// TIA Portal V20 export
FUNCTION_BLOCK "ErrComTextList"   // FB305, FBD
{ S7_Optimized_Access := 'TRUE' }
// stored: AutoNumber false, MemoryReserve 100, SetENOAutomatically false
   VAR
      Var { ExternalAccessible := 'False'; ExternalVisible := 'False'; ExternalWritable := 'False'} : "TypeVar";
      T { ExternalAccessible := 'False'; ExternalVisible := 'False'; ExternalWritable := 'False'} : Array[1..3] of IEC_TIMER;
      iLang { ExternalAccessible := 'False'; ExternalVisible := 'False'; ExternalWritable := 'False'} : Array[1..3] of DInt;
      sendImp { ExternalAccessible := 'False'; ExternalVisible := 'False'; ExternalWritable := 'False'} : Bool;
      sendTime { ExternalAccessible := 'False'; ExternalVisible := 'False'; ExternalWritable := 'False'} : Real;
      errNr { ExternalAccessible := 'False'; ExternalVisible := 'False'; ExternalWritable := 'False'} : DInt;
   END_VAR
   VAR_TEMP
      i : DInt;
      i2 : DInt;
      lowBound : DInt;
      upBound : DInt;
   END_VAR
BEGIN

REGION Network 1: sending impulse/clock
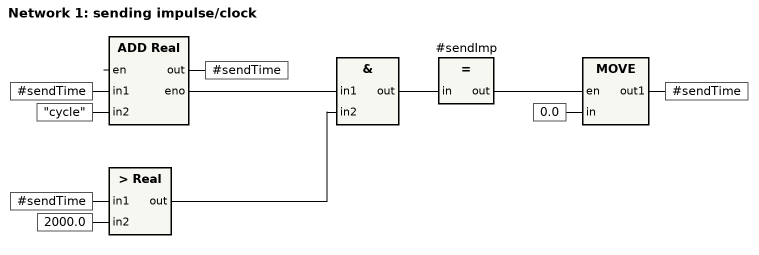
   #sendTime := #sendTime + "cycle";
   #sendImp := #sendTime > 2000.0;
   IF #sendImp THEN #sendTime := 0.0; END_IF;
END_REGION

REGION Network 2 (SCL): send step by step all the error list to Pc
   #lowBound := 2000;
   #upBound := 2205;

   IF #sendImp THEN

       #errNr += 1;
       IF #errNr > #upBound OR #errNr < #lowBound THEN
           #errNr := #lowBound;
       END_IF;

       "ComErrText".Sd.errList.idProd := 0;
       "ComErrText".Sd.errList.id := DINT_TO_UINT(#errNr);
       "ComErrText".Sd.errList.prio := "ErrTextList".err[#errNr].prio;
       "ComErrText".Sd.errList.timeStamp := DT_TO_LDT("Hmi".Clock.Act);

       #iLang[1] := #iLang[2] := #iLang[3] := 1;
       FOR #i := 1 TO 3 DO
           FOR #i2 := 1 TO 8 DO
               IF "ComErrText".Rd.language[#i] = "ErrTextList".language[#i2] AND "ComErrText".Rd.language[#i] <> WSTRING#'' THEN
                   #iLang[#i] := #i2;
                   EXIT;
               END_IF;
           END_FOR;
       END_FOR;

       "ComErrText".Sd.errList.alarm[1] := "ErrTextList".err[#errNr].alarm[#iLang[1]];
       "ComErrText".Sd.errList.info[1] := wstring#'';  
       "ComErrText".Sd.errList.remedy[1] := wstring#'';

       "ComErrText".Sd.errList.alarm[2] := "ErrTextList".err[#errNr].alarm[#iLang[2]];
       "ComErrText".Sd.errList.info[2] := wstring#'';
       "ComErrText".Sd.errList.remedy[2] := wstring#'';

       "ComErrText".Sd.errList.alarm[3] := "ErrTextList".err[#errNr].alarm[#iLang[3]];
       "ComErrText".Sd.errList.info[3] := wstring#'';
       "ComErrText".Sd.errList.remedy[3] := wstring#'';

   END_IF;
END_REGION
END_FUNCTION_BLOCK
